FUNCTION_BLOCK VisionStation EXTENDS MachineStation
VAR_INPUT
	rIO					: REFERENCE TO Vision_IO_typ;
	rStation			: REFERENCE TO Station;
	rKickoutStation 	: REFERENCE TO Station;
	rTrayLoadStation 	: REFERENCE TO Station;
END_VAR
VAR_OUTPUT
END_VAR
VAR
	Payload			: Payload_typ;
END_VAR

IF NOT (__ISVALIDREF(rStation) AND __ISVALIDREF(rIO) AND __ISVALIDREF(rKickoutStation) AND __ISVALIDREF(rTrayLoadStation)) THEN
	ADSLOGSTR( ADSLOG_MSGTYPE_ERROR, 'Invalid reference at %s.', InstancePath);	// how to make this work?
	RETURN;
END_IF

IF Enable THEN
	IF NOT _Enable THEN
		;
	END_IF

	CASE State OF
		STN_WAIT:
			IF Run AND rStation.MoverInPosition THEN
				State	:= STN_CHECKMOVER;
				Payload	:= rStation.CurrentMover.Payload;
			END_IF

		STN_CHECKMOVER:
				
			rIO.Outputs.Inspect := TRUE; // Start inspect
			
				
			
			IF rIO.Inputs.VisionActive THEN
				State := STN_PROCESS;
			END_IF

		STN_PROCESS:
			
				IF NOT(rIO.Inputs.VisionActive)THEN
					IF rIO.Inputs.VisionPass THEN
						Payload.VisionPass 	:= TRUE;
						
					ELSIF rIO.Inputs.VisionFail THEN
						Payload.VisionPass 	:= FALSE;
						
					ELSE // Failed to get feedback. TODO: Need alarm.
					END_IF;
					
					rIO.Outputs.Inspect := FALSE;
					State 				:= STN_SEND;
				END_IF;
					

		STN_SEND:
				
			IF Payload.VisionPass THEN
				rStation.CurrentMover.Payload	:= Payload;
				rStation.CurrentMover.MoveToStation(rTrayLoadStation);
				rStation.UnregisterCurrent();
			ELSE
				//Payload.Reject					:= TRUE;
				rStation.CurrentMover.Payload	:= Payload;
				rStation.CurrentMover.MoveToStation(rKickoutStation);
				rStation.UnregisterCurrent();
				
			END_IF;

			State							:= STN_WAIT;
		
		STN_ERROR:
	
	END_CASE

ELSIF _Enable THEN
	;
END_IF

//Save Previous Values
_Enable	:= Enable;

END_FUNCTION_BLOCK

(* stored: Version 1.1.0.1, ProductVersion 3.1.4024.12
   POU VisionStation: Id {7eb87a4f-bd9b-06c1-3178-f931d1986431}, SpecialFunc None *)
